FUNCTION_BLOCK GetVtcStatus (* Service Interface Block to read VT client status information using IsoVtcGetStatusInfo() *)
  (* Standard: ISO 11783-6; Description: Copyright (c) 2025 Meisterschulen am Ostbahnhof This program and the accompanying materials are made available under the terms of the Eclipse Public License 2.0 which is available at https://www.eclipse.org/legal/epl-2.0/ SPDX-License-Identifier: EPL-2.0 Service Interface Block to read VT client status information using IsoVtcGetStatusInfo() This block wraps the IsoVtcGetStatusInfo() function from the ISOBUS driver. It allows reading various status information about the VT client and connected VT. Available eVTInfo values (ISOVT_STATUS_e): - VT_SOURCE_ADDRESS (0): SA of VT - VT_HND (2): CF handle of VT - CF_SOURCE_ADDRESS (3): SA of VT client - CF_HND (4): CF handle of VT client - ID_VISIBLE_DATA_MASK (6): Data mask open on VT - ID_VISIBLE_SOFTKEY_MASK (7): Soft key mask open on VT - VT_BUSY_CODE (8): Busy code of VT Status message - AUXUNITS_TYPE1_ONBUS (9): ISO_TRUE if auxiliary unit type 1 is on bus - VT_ALIVE (11): VT lost for more than three seconds - VT_DOWNLOAD_FINISHED (12): Complete announcing finished - VT_POOL_ACTIVE_onVT (13): Pool active (selected) on VT - VT_STATEOFANNOUNCING (14): State of announcing - WS_VERSION_NR (15): Version number of working set - VT_NUMBOFVERSIONSTRINGS (16): Number of version strings sent of VT - VT_NAVSOFTKEYS (17): Navigation soft keys - Version 4 - VT_SOFTKEYXDOT (18): Softkey designator - pixel X - VT_SOFTKEYYDOT (19): Softkey designator - pixel Y - VT_VIRTUALSOFTKEYS (20): Number of virtual soft keys - VT_PHYSICALSOFTKEYS (21): Number of physical soft keys - VT_BOOTTIME (25): Boot time of VT - VT_GRAPHICTYPE (26): VT hardware - graphic type - VT_VERSIONNR (29): Version of working set VT *)
  (* Version 1.0, 2025-02-27, Generated, Meisterschulen am Ostbahnhof, initial API and implementation and/or initial documentation *)
  PACKAGE isobus::UT::status;
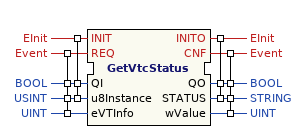
  EVENT_INPUT
    INIT : EInit WITH QI, u8Instance; (* Service Initialization *)
    REQ WITH QI, u8Instance, eVTInfo; (* Service Request - Read VT Status Info *)
  END_EVENT
  EVENT_OUTPUT
    INITO : EInit WITH QO, STATUS; (* Initialization Confirm *)
    CNF WITH QO, STATUS, wValue; (* Confirmation with result *)
  END_EVENT
  VAR_INPUT
    QI : BOOL; (* Quality Input - TRUE to enable service *)
    u8Instance : USINT; (* Identifier of the VT client instance (0-255) *)
    eVTInfo : UINT := 0; (* Status info type to read (ISOVT_STATUS_e enum value) *)
  END_VAR
  VAR_OUTPUT
    QO : BOOL; (* Quality Output - TRUE if service executed successfully *)
    STATUS : STRING; (* Service Status *)
    wValue : UINT; (* Returned status value from IsoVtcGetStatusInfo() *)
  END_VAR
END_FUNCTION_BLOCK
